{attribute 'linkalways'} 
{attribute 'no_explicit_call' := 'This FB is a CLASS and must be accessed using methods or properties'}
{attribute 'enable_dynamic_creation'}
FUNCTION_BLOCK Node_F_VN_ConvertPolarToCartesianPoints EXTENDS VisionNode
VAR
	ipSrcPointsPolar : _ITcVnContainer;
    ipDestPointsCart : _ITcVnContainer;
    hrPrev : _HRESULT(S_OK);
	hresult : _HRESULT(S_OK);
END_VAR

METHOD PUBLIC  Clone : I_Node
VAR
	pNode : POINTER TO Node_F_VN_ConvertPolarToCartesianPoints;
END_VAR
pNode := __NEW(Node_F_VN_ConvertPolarToCartesianPoints);
Clone := pNode^;
END_METHOD

METHOD FB_init : BOOL
VAR_INPUT
	bInitRetains : BOOL; // if TRUE, the retain variables are initialized (warm start / cold start)
	bInCopyCode : BOOL;  // if TRUE, the instance afterwards gets moved into the copy code (online change)
END_VAR
AddInput('ipSrcPointsPolar', ipSrcPointsPolar);
AddInput('hrPrev', hrPrev);
AddOutput('ipDestPointsCart', ipDestPointsCart);
AddOutput('hresult',hresult);
END_METHOD

METHOD PROTECTED OnExecute
hresult.Value := F_VN_ConvertPolarToCartesianPoints(
	ipSrcPointsPolar := ipSrcPointsPolar.Value,
	ipDestPointsCart := ipDestPointsCart.Value,
	hrPrev := hrPrev.Value);
END_METHOD

METHOD PUBLIC PreExecutionCheck
VAR_INPUT
	Check : I_PreExecutionChecks;
END_VAR
Check.IsTrue(ipSrcPointsPolar.IsValid, 'ipSrcPointsPolar must be a valid container');
Check.IsTrue((ipSrcPointsPolar.IsType(TC_GLOBAL_CONST_LIST.ContainerType_Vector_TcVnPoint2_REAL) OR
              ipSrcPointsPolar.IsType(TC_GLOBAL_CONST_LIST.ContainerType_Vector_TcVnPoint2_LREAL)),
              'ipSrcPointsPolar contains incorrect type');
END_METHOD

END_FUNCTION_BLOCK

(* stored: Version 1.1.0.1, ProductVersion 3.1.4026.13
   POU Node_F_VN_ConvertPolarToCartesianPoints: Id {45e67a53-7e89-0b8b-0ce1-bfc114bb1660}, SpecialFunc None
   Folder Constructor: Id {f27a62a9-e40c-076b-00e6-30542efaf256}
   Method Clone: Id {f4967600-5dd4-08c5-0dad-d24016ee58df}
   Method FB_init: Id {3d5992c1-68e5-0909-3f8b-3c5c64d7f548}
   Method OnExecute: Id {1499a784-2740-084f-05e5-13553e6cfbf8}
   Method PreExecutionCheck: Id {75807faa-1add-07f2-3976-a4fef4dbc6d7} *)
